TYPE
    ST_CSV_Line : STRUCT
        Fields : ARRAY[1..MAX_DATA_COUNT] OF T_MaxString;
    END_STRUCT
END_TYPE

(* stored: Version 1.1.0.1
   DUT ST_CSV_Line: Id {e6b5ba06-63b1-44fa-a491-2e87358904e4} *)
